{attribute 'GeneratedUsingTerminal: KL1002'}
{attribute addProperty BoxType "KL1002"}
{attribute addProperty Id "InputAT %I*BOOL0"}
{attribute addProperty CRC "2278121078"}
{attribute addProperty Size "0"}
TYPE Channel_87C95E76 :
STRUCT
	{attribute addProperty Name "Input"}
	Input AT %I* : BOOL;
END_STRUCT
END_TYPE

(* stored: Version 1.2.0.0, ProductVersion 3.1.4024.9
   DUT Channel_87C95E76: Id {a23b0bbc-789c-4189-990a-95ae8601875f} *)
